PROGRAM MAIN
VAR
	
	diStep : DINT;
	bStart : BOOL;
	bStop : BOOL;
	fbRepeatTimer : TON;
	udiCounter : UDINT;
	
	fbLogger : Logger:= (sPathName:='C:\Users\fboid\Documents\ScopeTest\Log.txt');
	fbNotifier : Notifier := (sPathName:='C:\Users\fboid\Documents\ScopeTest\Log.csv');
	fbNotifierEvent : NotifierEvent;
	i : INT;
	bExecute : BOOL;
	uiCounter : UINT:= 0;
	bMotorError : BOOL;
	
END_VAR

fbNotifier(bExecute := bExecute);
fbNotifierEvent(
	CLK:= bMotorError,  
	fbNotifier:= fbNotifier, 
	sModuleName := 'PreHeat',
	sDeviceName := 'Load conveyor',
	sStatus := 'Error',
	sMessage := 'Motor overloaded');

END_PROGRAM

(* stored: Version 1.1.0.1, ProductVersion 3.1.4024.2
   POU MAIN: Id {f62c6827-06de-4e99-83eb-58a9b7fb6cd1}, SpecialFunc None *)
